Yaskawa INFORM job: small_barrel_cylinder_program.JBI

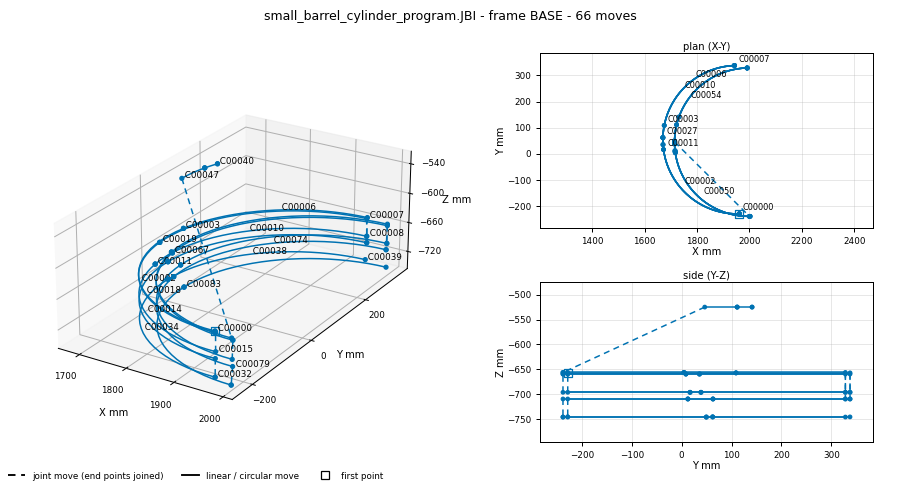
[picture p0: tool path of small_barrel_cylinder_program.JBI in frame BASE, 66 of 93 moves have a stored position in this frame; points joined in program order, loops and branches not executed]
/JOB
//NAME small_barrel_cylinder_program
//POS
///NPOS 88,0,88,0,0,0
///TOOL 0
///POSTYPE BASE
///RECTAN
///RCONF 0,0,0,0,0,0,0,0,0,0,0,0,0,0,0,0,0,0,0,0,0,0,0,0
C00000=1960.882173,-228.389361,-656.908500,-88.345417,-90.000000,5.000000
C00001=1960.882173,-228.389361,-656.908500,-88.345417,-90.000000,5.000000
C00002=1737.120796,-128.879052,-656.908500,-139.605563,-90.000000,5.000000
C00003=1674.905433,108.925066,-656.908500,168.928283,-89.999999,5.000000
C00004=1674.905433,108.925066,-656.908500,168.928283,-89.999999,5.000000
C00005=1674.905433,108.925066,-656.908500,168.928283,-89.999999,5.000000
C00006=1781.582896,280.054503,-656.908500,127.195122,-90.000000,5.000000
C00007=1943.333527,337.481320,-656.908500,91.897964,-90.000000,5.000000
C00008=1942.944258,337.468152,-695.836000,91.976800,-90.000000,5.000000
C00009=1942.944258,337.468152,-695.836000,91.976800,-90.000000,5.000000
C00010=1736.807224,237.639125,-695.836000,139.703600,-90.000000,5.000000
C00011=1672.166713,16.803437,-695.836000,-172.334018,-89.999999,5.000000
C00012=1672.166713,16.803437,-695.836000,-172.334018,-89.999999,5.000000
C00013=1672.166713,16.803437,-695.836000,-172.334018,-89.999999,5.000000
C00014=1771.103003,-162.573819,-695.836000,-129.907743,-90.000000,5.000000
C00015=1961.941112,-228.356789,-695.836000,-88.130979,-90.000000,5.000000
C00016=1961.917733,-228.357551,-659.247460,175.000000,-60.000000,91.864287
C00017=1961.917733,-228.357551,-659.247460,175.000000,-60.000000,91.864287
C00018=1770.798238,-162.318562,-659.247460,175.000000,-60.000000,50.011792
C00019=1670.264707,35.720420,-659.247460,-175.000000,-60.000000,5.000000
C00020=1670.264707,35.720420,-659.247460,-175.000000,-60.000000,5.000000
C00021=1670.264707,35.720420,-659.247460,-175.000000,-60.000000,5.000000
C00022=1739.257513,240.490177,-659.247460,175.000000,-60.000000,-41.057316
C00023=1941.902370,337.430270,-659.247460,175.000000,-60.000000,-87.812175
C00024=1943.337650,337.481457,-709.231960,175.000000,-60.000000,-88.102871
C00025=1943.337650,337.481457,-709.231960,175.000000,-60.000000,-88.102871
C00026=1754.177832,256.344745,-709.231960,175.000000,-60.000000,-45.465039
C00027=1669.755333,62.756374,-709.231960,175.000000,-60.000000,-5.000000
C00028=1669.755333,62.756374,-709.231960,175.000000,-60.000000,-5.000000
C00029=1669.755333,62.756374,-709.231960,175.000000,-60.000000,-5.000000
C00030=1748.422040,-141.386107,-709.231960,175.000000,-60.000000,43.806835
C00031=1961.183844,-228.380486,-709.231960,175.000000,-60.000000,91.715670
C00032=1960.709759,-228.394289,-745.172960,-175.000000,-60.000000,91.619671
C00033=1960.709759,-228.394289,-745.172960,-175.000000,-60.000000,91.619671
C00034=1749.673515,-142.682537,-745.172960,175.000000,-60.000000,44.171557
C00035=1669.737976,62.133101,-745.172960,175.000000,-60.000000,-5.000000
C00036=1669.737976,62.133101,-745.172960,175.000000,-60.000000,-5.000000
C00037=1669.737976,62.133101,-745.172960,175.000000,-60.000000,-5.000000
C00038=1740.751733,242.191820,-745.172960,-175.000000,-60.000000,-41.515683
C00039=1941.104098,337.398645,-745.172960,-175.000000,-60.000000,-87.650472
C00040=1730.919453,141.103894,-525.054000,160.183282,-90.000000,5.000000
C00041=1730.919453,141.103894,-525.054000,160.183282,-90.000000,5.000000
C00042=1725.296520,123.769589,-525.054000,163.872482,-90.000000,5.000000
C00043=1721.989762,111.270759,-525.054000,166.489602,-90.000000,5.000000
C00044=1721.989762,111.270759,-525.054000,166.489602,-90.000000,5.000000
C00045=1721.989762,111.270759,-525.054000,166.489602,-90.000000,5.000000
C00046=1714.467318,58.401379,-525.054000,175.000000,-90.000000,5.000000
C00047=1714.158726,46.270741,-525.054000,175.000000,-90.000000,5.000000
C00048=2000.218084,-237.917249,-656.077000,-89.394868,-90.000000,5.000000
C00049=2000.218084,-237.917249,-656.077000,-89.394868,-90.000000,5.000000
C00050=1810.535848,-167.641732,-656.077000,-131.263537,-90.000000,5.000000
C00051=1717.063414,4.675374,-656.077000,-171.781731,-90.000000,5.000000
C00052=1717.063414,4.675374,-656.077000,-171.781731,-90.000000,5.000000
C00053=1717.063414,4.675374,-656.077000,-171.781731,-90.000000,5.000000
C00054=1759.352323,198.581783,-656.077000,147.175822,-90.000000,5.000000
C00055=1991.673464,328.156453,-656.077000,91.124443,-90.000000,5.000000
C00056=1991.629264,328.155582,-695.827500,91.133392,-90.000000,5.000000
C00057=1991.629264,328.155582,-695.827500,91.133392,-90.000000,5.000000
C00058=1802.424600,250.519614,-695.827500,133.486038,-89.999999,5.000000
C00059=1714.230039,38.685390,-695.827500,-175.000000,-89.999999,5.000000
C00060=1714.230039,38.685390,-695.827500,-175.000000,-89.999999,5.000000
C00061=1714.230039,38.685390,-695.827500,-175.000000,-89.999999,5.000000
C00062=1797.728621,-155.683272,-695.827500,-134.810734,-90.000000,5.000000
C00063=2001.333786,-237.903266,-695.827500,-89.169024,-89.999999,5.000000
C00064=2002.654902,-237.881020,-659.230460,175.000000,-60.000000,91.098417
C00065=2002.654902,-237.881020,-659.230460,175.000000,-60.000000,91.098417
C00066=1816.210084,-172.489397,-659.230460,175.000000,-60.000000,50.247077
C00067=1716.545506,8.439722,-659.230460,175.000000,-60.000000,7.449155
C00068=1716.545506,8.439722,-659.230460,175.000000,-60.000000,7.449155
C00069=1716.545506,8.439722,-659.230460,175.000000,-60.000000,7.449155
C00070=1787.188756,234.910084,-659.230460,175.000000,-60.000000,-42.097850
C00071=1991.629329,328.155583,-659.230460,-175.000000,-60.000000,-88.866621
C00072=1990.432877,328.129382,-709.207960,-175.000000,-60.000000,-88.624393
C00073=1990.432877,328.129382,-709.207960,-175.000000,-60.000000,-88.624393
C00074=1789.492949,237.429663,-709.207960,175.000000,-60.000000,-42.788936
C00075=1716.049774,12.454082,-709.207960,-175.000000,-60.000000,6.630441
C00076=1716.049774,12.454082,-709.207960,-175.000000,-60.000000,6.630441
C00077=1716.049774,12.454082,-709.207960,-175.000000,-60.000000,6.630441
C00078=1809.884962,-167.068882,-709.207960,-175.000000,-60.000000,48.560962
C00079=2002.106712,-237.890999,-709.207960,-175.000000,-60.000000,90.987441
C00080=1999.227105,-237.925981,-745.458960,-175.000000,-60.000000,90.404543
C00081=1999.227105,-237.925981,-745.458960,-175.000000,-60.000000,90.404543
C00082=1784.013743,-141.057815,-745.458960,175.000000,-60.000000,41.130158
C00083=1714.189289,49.449706,-745.458960,175.000000,-60.000000,-5.000000
C00084=1714.189289,49.449706,-745.458960,175.000000,-60.000000,-5.000000
C00085=1714.189289,49.449706,-745.458960,175.000000,-60.000000,-5.000000
C00086=1788.890398,236.776662,-745.458960,175.000000,-60.000000,-42.609092
C00087=1991.442312,328.151821,-745.458960,175.000000,-60.000000,-88.828760
///POSTYPE PULSE
///PULSE
EX00000=94208.0
EX00001=277504.0
///POSTYPE PULSE
///PULSE
EC00000=94208.0
EC00001=94208.0
EC00002=94208.0
EC00003=94208.0
EC00004=94208.0
EC00005=94208.0
EC00006=94208.0
EC00007=94208.0
EC00008=94208.0
EC00009=94208.0
EC00010=94208.0
EC00011=94208.0
EC00012=94208.0
EC00013=94208.0
EC00014=94208.0
EC00015=94208.0
EC00016=94208.0
EC00017=94208.0
EC00018=94208.0
EC00019=94208.0
EC00020=94208.0
EC00021=94208.0
EC00022=94208.0
EC00023=94208.0
EC00024=94208.0
EC00025=94208.0
EC00026=94208.0
EC00027=94208.0
EC00028=94208.0
EC00029=94208.0
EC00030=94208.0
EC00031=94208.0
EC00032=94208.0
EC00033=94208.0
EC00034=94208.0
EC00035=94208.0
EC00036=94208.0
EC00037=94208.0
EC00038=94208.0
EC00039=94208.0
EC00040=277504.0
EC00041=277504.0
EC00042=277504.0
EC00043=277504.0
EC00044=277504.0
EC00045=277504.0
EC00046=277504.0
EC00047=277504.0
EC00048=277504.0
EC00049=277504.0
EC00050=277504.0
EC00051=277504.0
EC00052=277504.0
EC00053=277504.0
EC00054=277504.0
EC00055=277504.0
EC00056=277504.0
EC00057=277504.0
EC00058=277504.0
EC00059=277504.0
EC00060=277504.0
EC00061=277504.0
EC00062=277504.0
EC00063=277504.0
EC00064=277504.0
EC00065=277504.0
EC00066=277504.0
EC00067=277504.0
EC00068=277504.0
EC00069=277504.0
EC00070=277504.0
EC00071=277504.0
EC00072=277504.0
EC00073=277504.0
EC00074=277504.0
EC00075=277504.0
EC00076=277504.0
EC00077=277504.0
EC00078=277504.0
EC00079=277504.0
EC00080=277504.0
EC00081=277504.0
EC00082=277504.0
EC00083=277504.0
EC00084=277504.0
EC00085=277504.0
EC00086=277504.0
EC00087=277504.0
//INST
///DATE 2023/08/16 16:58
///ATTR SC,RW,RJ
////FRAME BASE
///GROUP1 RB1,ST1
NOP
MOVJ P009 EX000 VJ=15.00
MOVJ C00000 EC00000 VJ=15.0
CALL JOB:SPYON
MOVC C00001 EC00001 V=150.0
MOVC C00002 EC00002 V=150.0
MOVC C00003 EC00003 V=150.0
MOVJ C00004 EC00004 VJ=15.0
MOVC C00005 EC00005 V=150.0
MOVC C00006 EC00006 V=150.0
MOVC C00007 EC00007 V=150.0
MOVJ C00008 EC00008 VJ=15.0
MOVC C00009 EC00009 V=150.0
MOVC C00010 EC00010 V=150.0
MOVC C00011 EC00011 V=150.0
MOVJ C00012 EC00012 VJ=15.0
MOVC C00013 EC00013 V=150.0
MOVC C00014 EC00014 V=150.0
MOVC C00015 EC00015 V=150.0
MOVJ C00016 EC00016 VJ=15.0
MOVC C00017 EC00017 V=150.0
MOVC C00018 EC00018 V=150.0
MOVC C00019 EC00019 V=150.0
MOVJ C00020 EC00020 VJ=15.0
MOVC C00021 EC00021 V=150.0
MOVC C00022 EC00022 V=150.0
MOVC C00023 EC00023 V=150.0
MOVJ C00024 EC00024 VJ=15.0
MOVC C00025 EC00025 V=150.0
MOVC C00026 EC00026 V=150.0
MOVC C00027 EC00027 V=150.0
MOVJ C00028 EC00028 VJ=15.0
MOVC C00029 EC00029 V=150.0
MOVC C00030 EC00030 V=150.0
MOVC C00031 EC00031 V=150.0
MOVJ C00032 EC00032 VJ=15.0
MOVC C00033 EC00033 V=150.0
MOVC C00034 EC00034 V=150.0
MOVC C00035 EC00035 V=150.0
MOVJ C00036 EC00036 VJ=15.0
MOVC C00037 EC00037 V=150.0
MOVC C00038 EC00038 V=150.0
MOVC C00039 EC00039 V=150.0
CALL JOB:SPYOF
MOVJ P009 VJ=15.00
MOVL P009 EX00000 V=150.0
MOVJ C00040 EC00040 VJ=15.0
CALL JOB:SPYON
MOVC C00041 EC00041 V=150.0
MOVC C00042 EC00042 V=150.0
MOVC C00043 EC00043 V=150.0
MOVJ C00044 EC00044 VJ=15.0
MOVC C00045 EC00045 V=150.0
MOVC C00046 EC00046 V=150.0
MOVC C00047 EC00047 V=150.0
MOVJ C00048 EC00048 VJ=15.0
MOVC C00049 EC00049 V=150.0
MOVC C00050 EC00050 V=150.0
MOVC C00051 EC00051 V=150.0
MOVJ C00052 EC00052 VJ=15.0
MOVC C00053 EC00053 V=150.0
MOVC C00054 EC00054 V=150.0
MOVC C00055 EC00055 V=150.0
MOVJ C00056 EC00056 VJ=15.0
MOVC C00057 EC00057 V=150.0
MOVC C00058 EC00058 V=150.0
MOVC C00059 EC00059 V=150.0
MOVJ C00060 EC00060 VJ=15.0
MOVC C00061 EC00061 V=150.0
MOVC C00062 EC00062 V=150.0
MOVC C00063 EC00063 V=150.0
MOVJ C00064 EC00064 VJ=15.0
MOVC C00065 EC00065 V=150.0
MOVC C00066 EC00066 V=150.0
MOVC C00067 EC00067 V=150.0
MOVJ C00068 EC00068 VJ=15.0
MOVC C00069 EC00069 V=150.0
MOVC C00070 EC00070 V=150.0
MOVC C00071 EC00071 V=150.0
MOVJ C00072 EC00072 VJ=15.0
MOVC C00073 EC00073 V=150.0
MOVC C00074 EC00074 V=150.0
MOVC C00075 EC00075 V=150.0
MOVJ C00076 EC00076 VJ=15.0
MOVC C00077 EC00077 V=150.0
MOVC C00078 EC00078 V=150.0
MOVC C00079 EC00079 V=150.0
MOVJ C00080 EC00080 VJ=15.0
MOVC C00081 EC00081 V=150.0
MOVC C00082 EC00082 V=150.0
MOVC C00083 EC00083 V=150.0
MOVJ C00084 EC00084 VJ=15.0
MOVC C00085 EC00085 V=150.0
MOVC C00086 EC00086 V=150.0
MOVC C00087 EC00087 V=150.0
CALL JOB:SPYOF
MOVJ P009 VJ=15.00
MOVL P009 EX00001 V=150.0
END
